// TIA Portal V16 export
// export: Created 2024-05-10T06:46:44.3108547Z, ExportSetting WithDefaults, DisplayName Totally Integrated Automation Portal, DisplayVersion V16, DisplayName TIA Portal Version Control Interface, DisplayVersion V16, DisplayName TIA Portal Openness, DisplayVersion V16, DisplayName STEP 7 Professional, DisplayVersion V16, DisplayName STEP 7 Safety, DisplayVersion V16, DisplayName WinCC Professional, DisplayVersion V16
DATA_BLOCK "SinaParaS_DB"   // DB303
// stored: AutoNumber false, DBAccessibleFromOPCUA true, InstanceOfName SinaParaS, OfSystemLibElement SinaParaS, OfSystemLibVersion 1.0
"SinaParaS"
   // VAR_INPUT
   //    Start : Bool;
   //    ReadWrite : Bool;
   //    Parameter : Int;
   //    Index : Int;
   //    ValueWrite1 : Real;
   //    ValueWrite2 : DInt;
   //    AxisNo : Byte;
   //    hardwareId : HW_IO;
   // END_VAR
   // VAR_OUTPUT
   //    Ready : Bool;
   //    Busy : Bool;
   //    Done : Bool;
   //    ValueRead1 : Real;
   //    ValueRead2 : DInt;
   //    Format : Byte;
   //    ErrorNo : Word;
   //    Error : Bool;
   //    ErrorId : DWord;
   //    DiagId : Word;
   // END_VAR
   // VAR
   //    sbWrError : Bool;
   //    sbWrDone : Bool;
   //    sbRdError : Bool;
   //    sbWrBusy : Bool;
   //    sbRdBusy : Bool;
   //    sbWrStart : Bool;
   //    sbRdStart : Bool;
   //    sbWrStart1 : Bool;
   //    sbRdStart1 : Bool;
   //    sbWrStart2 : Bool;
   //    sbRdStart2 : Bool;
   //    sbStart : Bool;
   //    sbReady : Bool;
   //    sbRead : Bool;
   //    sbWrite : Bool;
   //    sbParaNo : Bool;
   //    sbBusy : Bool;
   //    sbError : Bool;
   //    sbDone : Bool;
   //    syFormat : Byte;
   //    syAxisNo : Byte;
   //    siReqRef : Int;
   //    siErrorId : Int;
   //    siErrorCount : Int;
   //    siMaxErrCount : Int;
   //    swParaError : Word;
   //    sReqParaMulti { S7_SetPoint := 'True'} : SinaReqPara;
   //    sChaParaMulti { S7_SetPoint := 'True'} : SinaChaPara;
   //    sRespParaMulti { S7_SetPoint := 'True'} : SinaRespPara;
   //    RDREC_1 { S7_SetPoint := 'True'} : RDREC;
   //    WRREC_1 { S7_SetPoint := 'True'} : WRREC;
   //    siLenHeader : Int;
   //    siLenParaMulti : Int;
   //    siLenChaPara : Int;
   // END_VAR
BEGIN
END_DATA_BLOCK
